// TIA Portal V19 export
FUNCTION "TEST_O_ACT_Fun" : Void   // FC206, LAD
// stored: SetENOAutomatically false
   VAR_TEMP   // added for the SCL form of the ladder/FBD networks
      _w1 : Bool;
   END_VAR
BEGIN

REGION Network 1
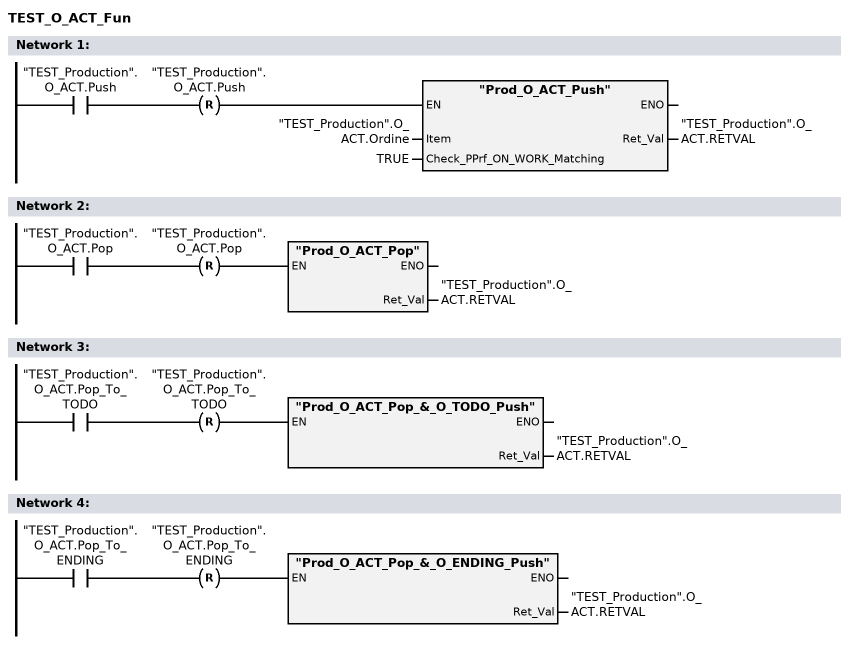
   RUNG wire#powerrail
      Contact( "TEST_Production".O_ACT.Push )
      R_Coil( "TEST_Production".O_ACT.Push )
      "Prod_O_ACT_Push"(Item := "TEST_Production".O_ACT.Ordine, Check_PPrf_ON_WORK_Matching := TRUE, Ret_Val => "TEST_Production".O_ACT.RETVAL)
   END_RUNG
   // the same network as SCL:
   #_w1 := "TEST_Production".O_ACT.Push;
   IF #_w1 THEN
       "TEST_Production".O_ACT.Push := FALSE;
       "TEST_Production".O_ACT.RETVAL := "Prod_O_ACT_Push"(Item := "TEST_Production".O_ACT.Ordine,
                               Check_PPrf_ON_WORK_Matching := TRUE);
   END_IF;
END_REGION

REGION Network 2
   RUNG wire#powerrail
      Contact( "TEST_Production".O_ACT.Pop )
      R_Coil( "TEST_Production".O_ACT.Pop )
      "Prod_O_ACT_Pop"(Ret_Val => "TEST_Production".O_ACT.RETVAL)
   END_RUNG
   // the same network as SCL:
   #_w1 := "TEST_Production".O_ACT.Pop;
   IF #_w1 THEN
       "TEST_Production".O_ACT.Pop := FALSE;
       "TEST_Production".O_ACT.RETVAL := "Prod_O_ACT_Pop"();
   END_IF;
END_REGION

REGION Network 3
   RUNG wire#powerrail
      Contact( "TEST_Production".O_ACT.Pop_To_TODO )
      R_Coil( "TEST_Production".O_ACT.Pop_To_TODO )
      "Prod_O_ACT_Pop_&_O_TODO_Push"(Ret_Val => "TEST_Production".O_ACT.RETVAL)
   END_RUNG
   // the same network as SCL:
   #_w1 := "TEST_Production".O_ACT.Pop_To_TODO;
   IF #_w1 THEN
       "TEST_Production".O_ACT.Pop_To_TODO := FALSE;
       "TEST_Production".O_ACT.RETVAL := "Prod_O_ACT_Pop_&_O_TODO_Push"();
   END_IF;
END_REGION

REGION Network 4
   RUNG wire#powerrail
      Contact( "TEST_Production".O_ACT.Pop_To_ENDING )
      R_Coil( "TEST_Production".O_ACT.Pop_To_ENDING )
      "Prod_O_ACT_Pop_&_O_ENDING_Push"(Ret_Val => "TEST_Production".O_ACT.RETVAL)
   END_RUNG
   // the same network as SCL:
   #_w1 := "TEST_Production".O_ACT.Pop_To_ENDING;
   IF #_w1 THEN
       "TEST_Production".O_ACT.Pop_To_ENDING := FALSE;
       "TEST_Production".O_ACT.RETVAL := "Prod_O_ACT_Pop_&_O_ENDING_Push"();
   END_IF;
END_REGION
END_FUNCTION
